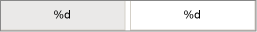
VISUALIZATION VISU_ConfigINTEntry  // 257x32
VAR_IN_OUT
    active : INT;
    editable : INT;
END_VAR
    Textfield (0,0 125x30), "%d", text variable: active, input disabled if: TRUE
    Textfield (130,0 125x30), "%d", text variable: editable, colour toggle: editable <> active
        OnMouseClick: write the text variable via Default
END_VISUALIZATION

(* stored: Version 1.1.0.1, ProductVersion 3.1.0.36
   Visu VISU_ConfigINTEntry: Id {77d57be9-9351-4a8f-a13b-c1958c674292} *)
